// TIA Portal V19 export
TYPE "LEXCHANGETRAY_typeSr1000ProfinetTelegram_operationinstructionControlBits"
// stored: Access Published
   STRUCT
      controlByte : Byte;
      readRequest : Bool;
      presetRequest : Bool;
      registerPresetDataReq : Bool;
      tuneRequest : Bool;
   END_STRUCT;
END_TYPE
